{attribute 'qualified_only'}
VAR_GLOBAL
Axes :  ARRAY[1..4] OF AXIS_REF;
END_VAR

(* stored: Version 1.1.0.1
   GVL GVL_Axes: Id {8ce01224-0deb-431a-815b-261aac9c5d7c} *)
